// TIA Portal project "Practica3AD21" (V16)

(* hardware
DEVICE "S7300/ET200M station_1"  S7-300 station
   slot 0: "Rail_0"  Rail  6ES7 390-1***0-0AA0
   slot 2: "PLC_1"  CPU 314  6ES7 314-1AG13-0AB0  V2.6
      slot 0: "MPI interface_1"  X1
*)

// ===== PLC "PLC_1"  CPU 314 =====

VAR_GLOBAL   // PLC tag table "Memorias"
   "E0" AT %M0.0 : Bool;   // Esperando a que haya pieza en almacen
   "E1" AT %M0.1 : Bool;   // Avanzando pieza
   "E2" AT %M0.2 : Bool;   // Primera ronda deteccion
   "E3" AT %M0.3 : Bool;   // Primera ronda ninguno
   "E4" AT %M0.4 : Bool;   // Primera ronda ambos
   "E5" AT %M0.5 : Bool;   // Primera ronda alguno
   "E6" AT %M0.6 : Bool;   // Pieza Tipo 1
   "E7" AT %M0.7 : Bool;   // Pieza Tipo 2
   "E8" AT %M1.0 : Bool;   // Pieza Tipo 3
   "E9" AT %M1.1 : Bool;   // Pieza Tipo 4
   "E10" AT %M1.6 : Bool;   // Extraer Piston 1
   "E11" AT %M1.7 : Bool;   // Extraer Piston 2
   "E12" AT %M2.0 : Bool;   // Extraer Piston 3
   "E13" AT %M2.1 : Bool;   // Contraer Piston 1
   "E14" AT %M2.2 : Bool;   // Contraer Piston 2
   "E15" AT %M2.3 : Bool;   // Contraer Piston 3
   "E16" AT %M2.4 : Bool;   // Pieza 1 Termina
   "E17" AT %M2.5 : Bool;   // Pieza 2 Termina
   "E18" AT %M2.6 : Bool;   // Pieza 3 Termina
   "E19" AT %M2.7 : Bool;   // Pieza 4 Termina
   "E20" AT %M3.0 : Bool;   // Detener Programa
END_VAR

VAR_GLOBAL   // PLC tag table "Salidas"
   "Chain" AT %Q11.0 : Bool;
   "Belt" AT %Q11.1 : Bool;
   "P1toWork" AT %Q11.2 : Bool;
   "P1toHome" AT %Q11.3 : Bool;
   "P2toWork" AT %Q11.4 : Bool;
   "P2toHome" AT %Q11.5 : Bool;
   "P3toWork" AT %Q11.6 : Bool;
   "P3toHome" AT %Q11.7 : Bool;
END_VAR

VAR_GLOBAL   // PLC tag table "Entradas"
   "P3inWork" AT %I10.0 : Bool;   // NC
   "P3inHome" AT %I10.1 : Bool;   // NC
   "P3engaged" AT %I10.2 : Bool;   // NO
   "RStation1" AT %I10.3 : Bool;   // NO
   "RStation2" AT %I10.4 : Bool;   // NO
   "Lightbarrier" AT %I10.5 : Bool;   // NC
   "inPlace3" AT %I10.6 : Bool;   // NO
   "inPlace4" AT %I10.7 : Bool;   // NO
   "P1inWork" AT %I11.0 : Bool;   // NC
   "P1inHome" AT %I11.1 : Bool;   // NC
   "P2inWork" AT %I11.2 : Bool;   // NC
   "P2inHome" AT %I11.3 : Bool;   // NC
   "P1engaged" AT %I11.4 : Bool;   // NO
   "P2engaged" AT %I11.5 : Bool;   // NO
   "inPlace1" AT %I11.6 : Bool;   // NO
   "inPlace2" AT %I11.7 : Bool;   // NO
   "chainMagnet" AT %I13.6 : Bool;   // NO
   "STOP" AT %I13.7 : Bool;   // NO
   "START" AT %I13.5 : Bool;   // NO
END_VAR

// folder: SystemBlocksFolder/ReportSystemErrorFolder

DATA_BLOCK "RSE_DIAGNOSTIC_STATUS_DB"   // DB127
TITLE = Report System Error Diagnostic Block
{ S7_Optimized_Access := 'FALSE' }
AUTHOR : SIMATIC
FAMILY : RSEDIAG
NAME : RSE7
VERSION : 1.0
// This DB is part of report system error and will be updated by the RSE FB.
//  It is an interface for support of system diagnosis via the CPU web server.
   VAR
      Directory : Struct
         D_Version : Word := WORD#16#0100;   // Version that supports RSE
         D_pGlobalState : Word := WORD#16#0010;   // Byte offset to the start of the "GlobalState" section
         D_pQuery : Word := WORD#16#0014;   // Byte offset to the start of the "Query" section
         D_pComponent : Word := WORD#16#0020;   // Byte offset to the start of the "Component" section
         D_pError : Word := WORD#16#0024;   // Byte offset to the start of the "Error" section
         D_pState : Word := WORD#16#0028;   // Byte offset to the start of the "State" section
         D_pAlarm : Word := WORD#16#005A;   // Byte offset to the start of the "Alarm" section
         D_pSubComponent : Word := WORD#16#0082;   // Byte offset to the start of the "Subcomponent" section
      END_STRUCT;
      GlobalState : Struct
         G_EventCount : Word := WORD#16#0000;   // ID of the last event (counter)
         G_StartReporting : Bool := FALSE;   // Startup evaluation running
      END_STRUCT;
      Query : Struct
         Q_ClientID_User : DWord := DWORD#16#0000_0000;   // ID of the client
         Q_ClientID_Intern : DWord := DWORD#16#0000_0000;   // ID of the client (internal)
         Q_WithSubComponent : Bool := FALSE;   // With/without status of the underlying components (slower)
         Q_SubComponentAlarm : Bool := FALSE;   // AS-iMaster gibt AS-iSlave Alarme zurück
         Q_Reserved2 : Bool := FALSE;   // Reserved
         Q_Reserved3 : Bool := FALSE;   // Reserved
         Q_Reserved4 : Bool := FALSE;   // Reserved
         Q_Reserved5 : Bool := FALSE;   // Reserved
         Q_Reserved6 : Bool := FALSE;   // Reserved
         Q_Reserved7 : Bool := FALSE;   // Reserved
         Q_Start : Bool := FALSE;   // Start query
         Q_Error : Byte := BYTE#16#00;   // Internal error in query
         Q_Reserved8 : Byte := BYTE#16#00;   // Reserved
      END_STRUCT;
      Component : Struct
         C_AddressMode : Byte := BYTE#16#00;   // Addressing mode of the module
         C_Reserved1 : Byte := BYTE#16#00;   // Reserved
         C_ComponentID : Word := WORD#16#0000;   // Hardware ID of the component (internal)
      END_STRUCT;
      Error : Struct
         E_ErrorNo : Word := WORD#16#0000;   // Index of the requested/actual error
         E_LastError : Bool := FALSE;   // TRUE, if E_ErrorNo contains the indes of the last error, otherwise FALSE
      END_STRUCT;
      State : Struct
         S_Hierarchy : Byte := BYTE#16#00;   // Reserved
         S_Periphery : Byte := BYTE#16#00;   // Reserved
         S_SupFault : Bool := FALSE;   // The component is not obtainable
         S_NotAvailable : Bool := FALSE;   // The component does not exist
         S_Faulty : Bool := FALSE;   // The component is disrupted; the "Alarm" section is not empty
         S_MoreErrors : Bool := FALSE;   // There are more errors than RSE can store.
         S_Maintenance1 : Bool := FALSE;   // Maintenance required is indicated
         S_Maintenance2 : Bool := FALSE;   // Maintenance demand is indicated
         S_Deactivated : Bool := FALSE;   // The component was deactivated
         S_Reserved2 : Bool := FALSE;   // Reserved
         S_SubFault : Bool := FALSE;   // An underlying component is disrupted
         S_SubMaintenance1 : Bool := FALSE;   // Maintenance required is indicated for an underlying component
         S_SubMaintenance2 : Bool := FALSE;   // Maintenance demand is indicated for an underlying component
         S_SubDeactivated : Bool := FALSE;   // At least one lower-level component is disabled
         S_Reserved4 : Bool := FALSE;   // Reserved
         S_Reserved5 : Bool := FALSE;   // Reserved
         S_Reserved6 : Bool := FALSE;   // Reserved
         S_Reserved7 : Bool := FALSE;   // Reserved
         S_TIAMS : DWord := DWORD#16#0000_0000;   // Maintenance state of the component
         S_TIAMSChannelExist : DWord := DWORD#16#0000_0000;   // Maintenance state: Configured channels
         S_TIAMSChannelOK : DWord := DWORD#16#0000_0000;   // Maintenance State: Disrupted channels
         S_ChannelCount : Word := WORD#16#0000;   // Number of channels; Valid only when Q_WithSubComponent is set
         S_ChannelVector : Array[0..255] of Bool;   // List of channels involved; Valid only when Q_WithSubComponent is set
      END_STRUCT;
      Alarm : Struct
         A_ComponentID : Word := WORD#16#0000;   // Hardware ID of the component (internal)
         A_TextID1 : Word := WORD#16#0000;   // ID of the first error text
         A_TextLexikonID1 : Word := WORD#16#0000;   // ID of the first error text lexicon
         A_HelpTextLexikonID1 : Word := WORD#16#0000;   // ID of the first help text lexicon
         A_MapTextID : Word := WORD#16#0000;   // ID of the first error text in the export file (HMI)
         A_MapHelpTextID : Word := WORD#16#0000;   // ID of the first help text in the export file (HMI)
         A_TextID2 : Word := WORD#16#0000;   // ID of the second error text
         A_TextLexikonID2 : Word := WORD#16#0000;   // ID of the second error text lexicon
         A_HelpTextLexikonID2 : Word := WORD#16#0000;   // ID of the second help text lexicon
         A_MapTextID2 : Word := WORD#16#0000;   // ID of the second error text in the export file (HMI)
         A_MapHelpTextID2 : Word := WORD#16#0000;   // ID of the second help text in the export file (HMI)
         A_AlarmID : DWord := DWORD#16#0000_0000;   // Message number
         A_ValueCount : Word := WORD#16#000C;   // Number of other occupied bytes
         A_AssociatedValue : Array[1..6] of Word;   // Associated values of the message
      END_STRUCT;
      SubComponent : Struct
         U_SubComponentCount : Word := WORD#16#0000;   // Number of underlying components
         U_SubComponentFault : Array[1..4] of Byte;   // List of status of subordinate components, 1 byte per component
      END_STRUCT;
   END_VAR
BEGIN
END_DATA_BLOCK

// folder: (top level)

FUNCTION "Secuencial" : Void   // FC1, LAD
{ S7_Optimized_Access := 'FALSE' }
VERSION : 0.1
   VAR_TEMP
      T1A : Time;
   END_VAR
   VAR_TEMP   // added for the SCL form of the ladder/FBD networks
      _w1 : Bool;
   END_VAR
BEGIN

REGION Network 1: Avanzando pieza
   // Si se detecta una pieza en el almacen y no se ha apretado STOP, mover la cadena
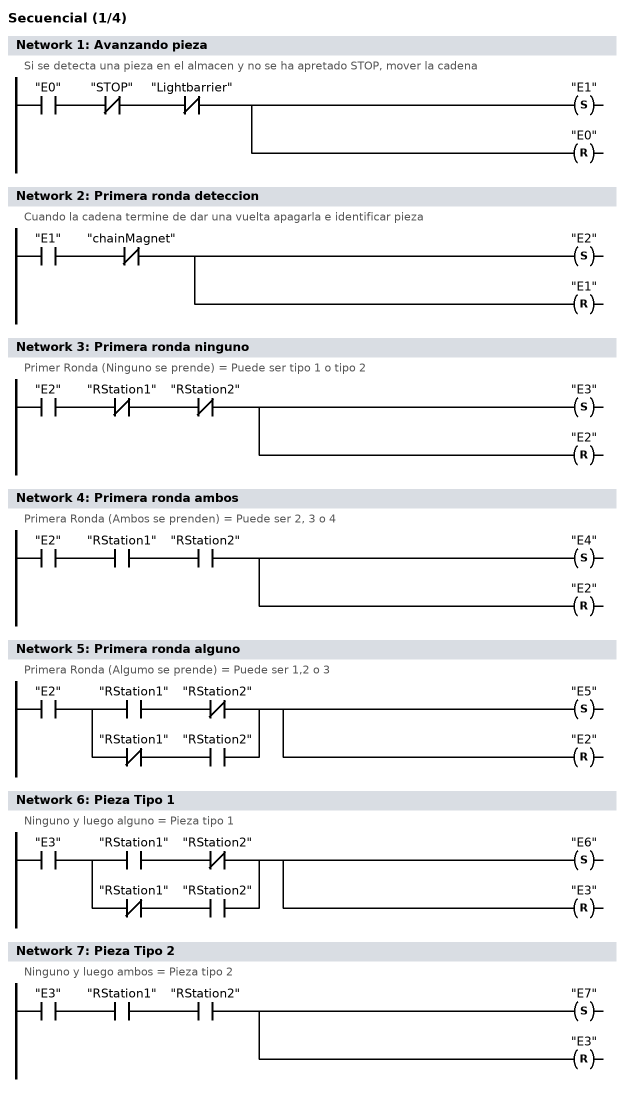
   RUNG wire#powerrail
      Contact( "E0" )
      I_Contact( "STOP" )
      I_Contact( "Lightbarrier" )
      wire#w1
      S_Coil( "E1" )
   END_RUNG
   RUNG wire#w1
      R_Coil( "E0" )
   END_RUNG
   // the same network as SCL:
   IF "E0" AND NOT "STOP" AND NOT "Lightbarrier" THEN
       "E1" := TRUE;
       "E0" := FALSE;
   END_IF;
END_REGION

REGION Network 2: Primera ronda deteccion
   // Cuando la cadena termine de dar una vuelta apagarla e identificar pieza
   RUNG wire#powerrail
      Contact( "E1" )
      I_Contact( "chainMagnet" )
      wire#w1
      S_Coil( "E2" )
   END_RUNG
   RUNG wire#w1
      R_Coil( "E1" )
   END_RUNG
   // the same network as SCL:
   IF "E1" AND NOT "chainMagnet" THEN
       "E2" := TRUE;
       "E1" := FALSE;
   END_IF;
END_REGION

REGION Network 3: Primera ronda ninguno
   // Primer Ronda (Ninguno se prende) = Puede ser tipo 1 o tipo 2
   RUNG wire#powerrail
      Contact( "E2" )
      I_Contact( "RStation1" )
      I_Contact( "RStation2" )
      wire#w1
      S_Coil( "E3" )
   END_RUNG
   RUNG wire#w1
      R_Coil( "E2" )
   END_RUNG
   // the same network as SCL:
   IF "E2" AND NOT "RStation1" AND NOT "RStation2" THEN
       "E3" := TRUE;
       "E2" := FALSE;
   END_IF;
END_REGION

REGION Network 4: Primera ronda ambos
   // Primera Ronda (Ambos se prenden) = Puede ser 2, 3 o 4
   RUNG wire#powerrail
      Contact( "E2" )
      Contact( "RStation1" )
      Contact( "RStation2" )
      wire#w1
      S_Coil( "E4" )
   END_RUNG
   RUNG wire#w1
      R_Coil( "E2" )
   END_RUNG
   // the same network as SCL:
   IF "E2" AND "RStation1" AND "RStation2" THEN
       "E4" := TRUE;
       "E2" := FALSE;
   END_IF;
END_REGION

REGION Network 5: Primera ronda alguno
   // Primera Ronda (Algumo se prende) = Puede ser 1,2 o 3
   RUNG wire#powerrail
      Contact( "E2" )
      wire#w1
      Contact( "RStation1" )
      I_Contact( "RStation2" )
      wire#w2
      S_Coil( "E5" )
   END_RUNG
   RUNG wire#w1
      I_Contact( "RStation1" )
      Contact( "RStation2" )
   END_RUNG wire#w2
   RUNG wire#w2
      R_Coil( "E2" )
   END_RUNG
   // the same network as SCL:
   IF "E2" AND (("RStation1" AND NOT "RStation2") OR (NOT "RStation1" AND "RStation2")) THEN
       "E5" := TRUE;
       "E2" := FALSE;
   END_IF;
END_REGION

REGION Network 6: Pieza Tipo 1
   // Ninguno y luego alguno = Pieza tipo 1
   RUNG wire#powerrail
      Contact( "E3" )
      wire#w1
      Contact( "RStation1" )
      I_Contact( "RStation2" )
      wire#w2
      S_Coil( "E6" )
   END_RUNG
   RUNG wire#w1
      I_Contact( "RStation1" )
      Contact( "RStation2" )
   END_RUNG wire#w2
   RUNG wire#w2
      R_Coil( "E3" )
   END_RUNG
   // the same network as SCL:
   IF "E3" AND (("RStation1" AND NOT "RStation2") OR (NOT "RStation1" AND "RStation2")) THEN
       "E6" := TRUE;
       "E3" := FALSE;
   END_IF;
END_REGION

REGION Network 7: Pieza Tipo 2
   // Ninguno y luego ambos = Pieza tipo 2
   RUNG wire#powerrail
      Contact( "E3" )
      Contact( "RStation1" )
      Contact( "RStation2" )
      wire#w1
      S_Coil( "E7" )
   END_RUNG
   RUNG wire#w1
      R_Coil( "E3" )
   END_RUNG
   // the same network as SCL:
   IF "E3" AND "RStation1" AND "RStation2" THEN
       "E7" := TRUE;
       "E3" := FALSE;
   END_IF;
END_REGION

REGION Network 8: Pieza Tipo 2
   // Ambos y luego ninguno = Pieza tipo 2
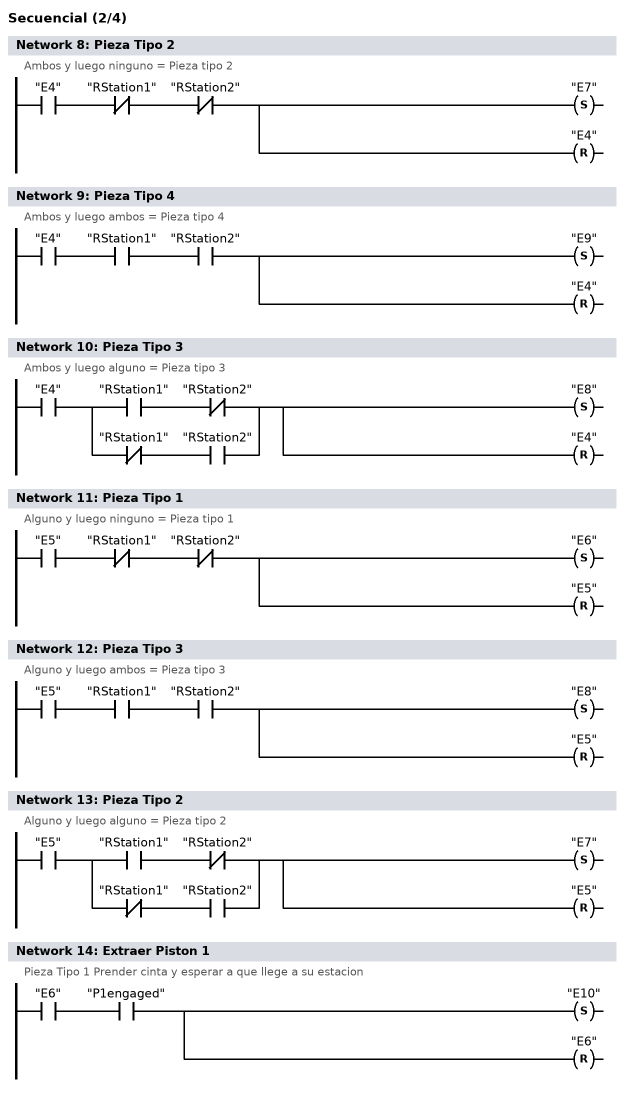
   RUNG wire#powerrail
      Contact( "E4" )
      I_Contact( "RStation1" )
      I_Contact( "RStation2" )
      wire#w1
      S_Coil( "E7" )
   END_RUNG
   RUNG wire#w1
      R_Coil( "E4" )
   END_RUNG
   // the same network as SCL:
   IF "E4" AND NOT "RStation1" AND NOT "RStation2" THEN
       "E7" := TRUE;
       "E4" := FALSE;
   END_IF;
END_REGION

REGION Network 9: Pieza Tipo 4
   // Ambos y luego ambos = Pieza tipo 4
   RUNG wire#powerrail
      Contact( "E4" )
      Contact( "RStation1" )
      Contact( "RStation2" )
      wire#w1
      S_Coil( "E9" )
   END_RUNG
   RUNG wire#w1
      R_Coil( "E4" )
   END_RUNG
   // the same network as SCL:
   IF "E4" AND "RStation1" AND "RStation2" THEN
       "E9" := TRUE;
       "E4" := FALSE;
   END_IF;
END_REGION

REGION Network 10: Pieza Tipo 3
   // Ambos y luego alguno = Pieza tipo 3
   RUNG wire#powerrail
      Contact( "E4" )
      wire#w1
      Contact( "RStation1" )
      I_Contact( "RStation2" )
      wire#w2
      S_Coil( "E8" )
   END_RUNG
   RUNG wire#w1
      I_Contact( "RStation1" )
      Contact( "RStation2" )
   END_RUNG wire#w2
   RUNG wire#w2
      R_Coil( "E4" )
   END_RUNG
   // the same network as SCL:
   IF "E4" AND (("RStation1" AND NOT "RStation2") OR (NOT "RStation1" AND "RStation2")) THEN
       "E8" := TRUE;
       "E4" := FALSE;
   END_IF;
END_REGION

REGION Network 11: Pieza Tipo 1
   // Alguno y luego ninguno = Pieza tipo 1
   RUNG wire#powerrail
      Contact( "E5" )
      I_Contact( "RStation1" )
      I_Contact( "RStation2" )
      wire#w1
      S_Coil( "E6" )
   END_RUNG
   RUNG wire#w1
      R_Coil( "E5" )
   END_RUNG
   // the same network as SCL:
   IF "E5" AND NOT "RStation1" AND NOT "RStation2" THEN
       "E6" := TRUE;
       "E5" := FALSE;
   END_IF;
END_REGION

REGION Network 12: Pieza Tipo 3
   // Alguno y luego ambos = Pieza tipo 3
   RUNG wire#powerrail
      Contact( "E5" )
      Contact( "RStation1" )
      Contact( "RStation2" )
      wire#w1
      S_Coil( "E8" )
   END_RUNG
   RUNG wire#w1
      R_Coil( "E5" )
   END_RUNG
   // the same network as SCL:
   IF "E5" AND "RStation1" AND "RStation2" THEN
       "E8" := TRUE;
       "E5" := FALSE;
   END_IF;
END_REGION

REGION Network 13: Pieza Tipo 2
   // Alguno y luego alguno = Pieza tipo 2
   RUNG wire#powerrail
      Contact( "E5" )
      wire#w1
      Contact( "RStation1" )
      I_Contact( "RStation2" )
      wire#w2
      S_Coil( "E7" )
   END_RUNG
   RUNG wire#w1
      I_Contact( "RStation1" )
      Contact( "RStation2" )
   END_RUNG wire#w2
   RUNG wire#w2
      R_Coil( "E5" )
   END_RUNG
   // the same network as SCL:
   IF "E5" AND (("RStation1" AND NOT "RStation2") OR (NOT "RStation1" AND "RStation2")) THEN
       "E7" := TRUE;
       "E5" := FALSE;
   END_IF;
END_REGION

REGION Network 14: Extraer Piston 1
   // Pieza Tipo 1 Prender cinta y esperar a que llege a su estacion
   RUNG wire#powerrail
      Contact( "E6" )
      Contact( "P1engaged" )
      wire#w1
      S_Coil( "E10" )
   END_RUNG
   RUNG wire#w1
      R_Coil( "E6" )
   END_RUNG
   // the same network as SCL:
   IF "E6" AND "P1engaged" THEN
       "E10" := TRUE;
       "E6" := FALSE;
   END_IF;
END_REGION

REGION Network 15: Extraer Piston 2
   // Pieza Tipo 2 Prender cinta y esperar a que llege a su estacion
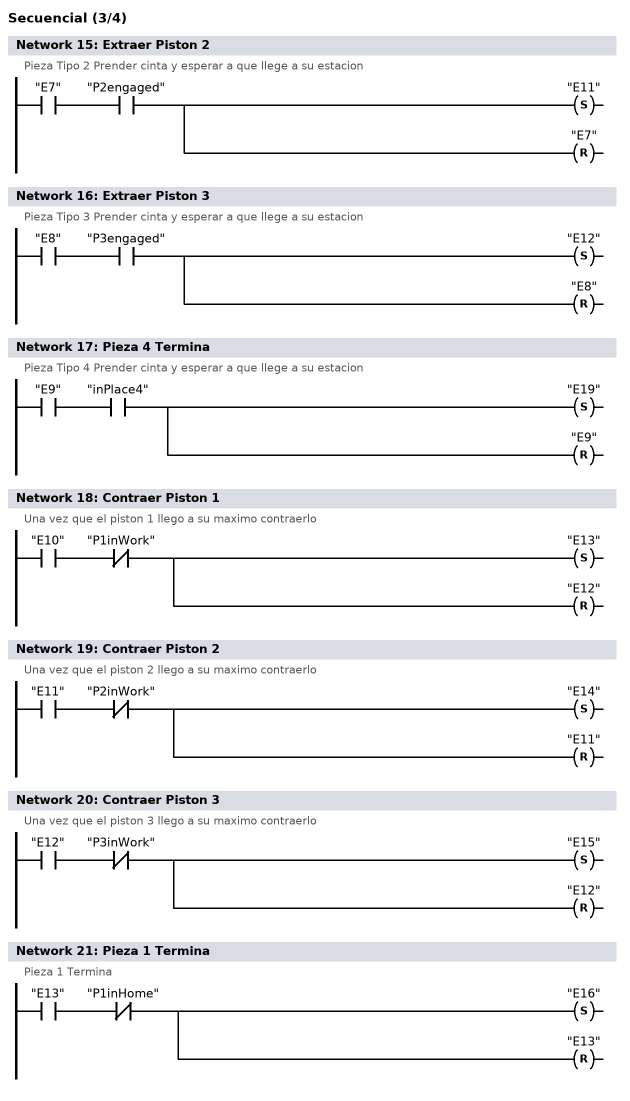
   RUNG wire#powerrail
      Contact( "E7" )
      Contact( "P2engaged" )
      wire#w1
      S_Coil( "E11" )
   END_RUNG
   RUNG wire#w1
      R_Coil( "E7" )
   END_RUNG
   // the same network as SCL:
   IF "E7" AND "P2engaged" THEN
       "E11" := TRUE;
       "E7" := FALSE;
   END_IF;
END_REGION

REGION Network 16: Extraer Piston 3
   // Pieza Tipo 3 Prender cinta y esperar a que llege a su estacion
   RUNG wire#powerrail
      Contact( "E8" )
      Contact( "P3engaged" )
      wire#w1
      S_Coil( "E12" )
   END_RUNG
   RUNG wire#w1
      R_Coil( "E8" )
   END_RUNG
   // the same network as SCL:
   IF "E8" AND "P3engaged" THEN
       "E12" := TRUE;
       "E8" := FALSE;
   END_IF;
END_REGION

REGION Network 17: Pieza 4 Termina
   // Pieza Tipo 4 Prender cinta y esperar a que llege a su estacion
   RUNG wire#powerrail
      Contact( "E9" )
      Contact( "inPlace4" )
      wire#w1
      S_Coil( "E19" )
   END_RUNG
   RUNG wire#w1
      R_Coil( "E9" )
   END_RUNG
   // the same network as SCL:
   IF "E9" AND "inPlace4" THEN
       "E19" := TRUE;
       "E9" := FALSE;
   END_IF;
END_REGION

REGION Network 18: Contraer Piston 1
   // Una vez que el piston 1 llego a su maximo contraerlo
   RUNG wire#powerrail
      Contact( "E10" )
      I_Contact( "P1inWork" )
      wire#w1
      S_Coil( "E13" )
   END_RUNG
   RUNG wire#w1
      R_Coil( "E12" )
   END_RUNG
   // the same network as SCL:
   IF "E10" AND NOT "P1inWork" THEN
       "E13" := TRUE;
       "E12" := FALSE;
   END_IF;
END_REGION

REGION Network 19: Contraer Piston 2
   // Una vez que el piston 2 llego a su maximo contraerlo
   RUNG wire#powerrail
      Contact( "E11" )
      I_Contact( "P2inWork" )
      wire#w1
      S_Coil( "E14" )
   END_RUNG
   RUNG wire#w1
      R_Coil( "E11" )
   END_RUNG
   // the same network as SCL:
   IF "E11" AND NOT "P2inWork" THEN
       "E14" := TRUE;
       "E11" := FALSE;
   END_IF;
END_REGION

REGION Network 20: Contraer Piston 3
   // Una vez que el piston 3 llego a su maximo contraerlo
   RUNG wire#powerrail
      Contact( "E12" )
      I_Contact( "P3inWork" )
      wire#w1
      S_Coil( "E15" )
   END_RUNG
   RUNG wire#w1
      R_Coil( "E12" )
   END_RUNG
   // the same network as SCL:
   IF "E12" AND NOT "P3inWork" THEN
       "E15" := TRUE;
       "E12" := FALSE;
   END_IF;
END_REGION

REGION Network 21: Pieza 1 Termina
   // Pieza 1 Termina
   RUNG wire#powerrail
      Contact( "E13" )
      I_Contact( "P1inHome" )
      wire#w1
      S_Coil( "E16" )
   END_RUNG
   RUNG wire#w1
      R_Coil( "E13" )
   END_RUNG
   // the same network as SCL:
   IF "E13" AND NOT "P1inHome" THEN
       "E16" := TRUE;
       "E13" := FALSE;
   END_IF;
END_REGION

REGION Network 22: Pieza 2 Termina
   // Pieza 2 Termina
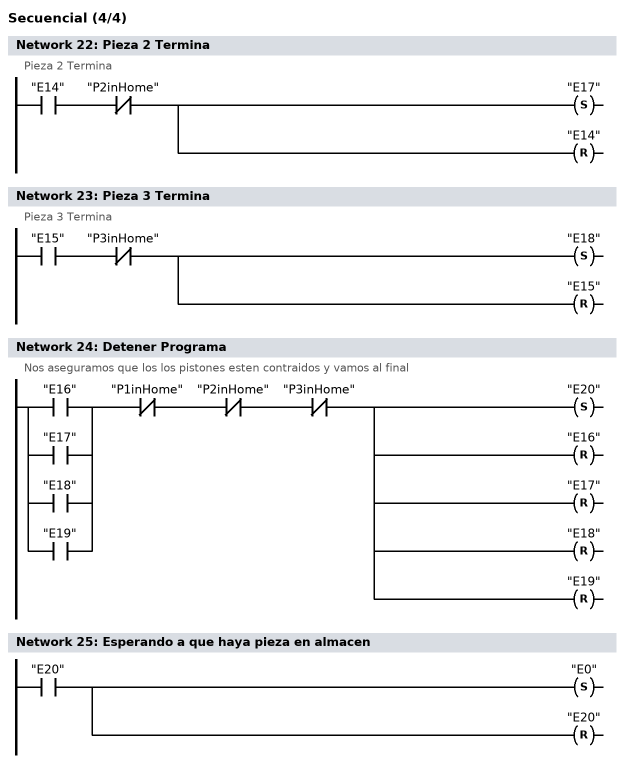
   RUNG wire#powerrail
      Contact( "E14" )
      I_Contact( "P2inHome" )
      wire#w1
      S_Coil( "E17" )
   END_RUNG
   RUNG wire#w1
      R_Coil( "E14" )
   END_RUNG
   // the same network as SCL:
   IF "E14" AND NOT "P2inHome" THEN
       "E17" := TRUE;
       "E14" := FALSE;
   END_IF;
END_REGION

REGION Network 23: Pieza 3 Termina
   // Pieza 3 Termina
   RUNG wire#powerrail
      Contact( "E15" )
      I_Contact( "P3inHome" )
      wire#w1
      S_Coil( "E18" )
   END_RUNG
   RUNG wire#w1
      R_Coil( "E15" )
   END_RUNG
   // the same network as SCL:
   IF "E15" AND NOT "P3inHome" THEN
       "E18" := TRUE;
       "E15" := FALSE;
   END_IF;
END_REGION

REGION Network 24: Detener Programa
   // Nos aseguramos que los los pistones esten contraidos y vamos al final
   RUNG wire#powerrail
      Contact( "E16" )
      wire#w1
      I_Contact( "P1inHome" )
      I_Contact( "P2inHome" )
      I_Contact( "P3inHome" )
      wire#w2
      S_Coil( "E20" )
   END_RUNG
   RUNG wire#powerrail
      Contact( "E17" )
   END_RUNG wire#w1
   RUNG wire#powerrail
      Contact( "E18" )
   END_RUNG wire#w1
   RUNG wire#powerrail
      Contact( "E19" )
   END_RUNG wire#w1
   RUNG wire#w2
      R_Coil( "E16" )
   END_RUNG
   RUNG wire#w2
      R_Coil( "E17" )
   END_RUNG
   RUNG wire#w2
      R_Coil( "E18" )
   END_RUNG
   RUNG wire#w2
      R_Coil( "E19" )
   END_RUNG
   // the same network as SCL:
   IF ("E16" OR "E17" OR "E18" OR "E19") AND NOT "P1inHome" AND NOT "P2inHome" AND NOT "P3inHome" THEN
       "E20" := TRUE;
   END_IF;
   #_w1 := ("E16" OR "E17" OR "E18" OR "E19") AND NOT "P1inHome" AND NOT "P2inHome" AND NOT "P3inHome";
   IF #_w1 THEN
       "E16" := FALSE;
       "E17" := FALSE;
       "E18" := FALSE;
       "E19" := FALSE;
   END_IF;
END_REGION

REGION Network 25: Esperando a que haya pieza en almacen
   RUNG wire#powerrail
      Contact( "E20" )
      wire#w1
      S_Coil( "E0" )
   END_RUNG
   RUNG wire#w1
      R_Coil( "E20" )
   END_RUNG
   // the same network as SCL:
   IF "E20" THEN
       "E0" := TRUE;
       "E20" := FALSE;
   END_IF;
END_REGION
END_FUNCTION

FUNCTION "Combinacional" : Void   // FC2, LAD
{ S7_Optimized_Access := 'FALSE' }
VERSION : 0.1
BEGIN

REGION Network 1
   // Cuando inicia el programa todo esta apagado
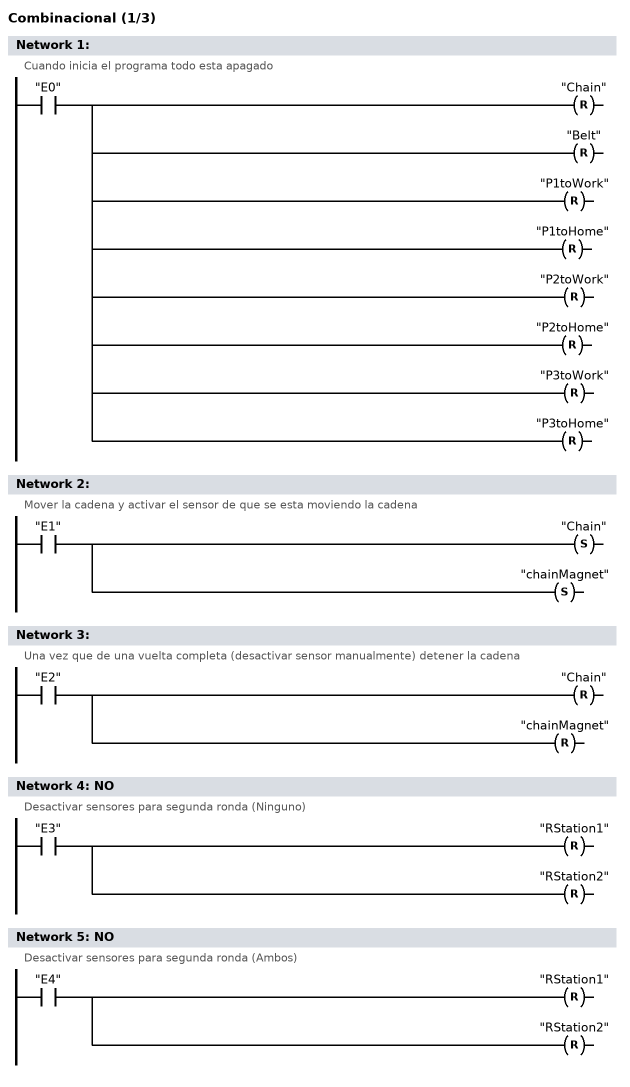
   RUNG wire#powerrail
      Contact( "E0" )
      wire#w1
      R_Coil( "Chain" )
   END_RUNG
   RUNG wire#w1
      R_Coil( "Belt" )
   END_RUNG
   RUNG wire#w1
      R_Coil( "P1toWork" )
   END_RUNG
   RUNG wire#w1
      R_Coil( "P1toHome" )
   END_RUNG
   RUNG wire#w1
      R_Coil( "P2toWork" )
   END_RUNG
   RUNG wire#w1
      R_Coil( "P2toHome" )
   END_RUNG
   RUNG wire#w1
      R_Coil( "P3toWork" )
   END_RUNG
   RUNG wire#w1
      R_Coil( "P3toHome" )
   END_RUNG
   // the same network as SCL:
   IF "E0" THEN
       "Chain" := FALSE;
       "Belt" := FALSE;
       "P1toWork" := FALSE;
       "P1toHome" := FALSE;
       "P2toWork" := FALSE;
       "P2toHome" := FALSE;
       "P3toWork" := FALSE;
       "P3toHome" := FALSE;
   END_IF;
END_REGION

REGION Network 2
   // Mover la cadena y activar el sensor de que se esta moviendo la cadena
   RUNG wire#powerrail
      Contact( "E1" )
      wire#w1
      S_Coil( "Chain" )
   END_RUNG
   RUNG wire#w1
      S_Coil( "chainMagnet" )
   END_RUNG
   // the same network as SCL:
   IF "E1" THEN
       "Chain" := TRUE;
       "chainMagnet" := TRUE;
   END_IF;
END_REGION

REGION Network 3
   // Una vez que de una vuelta completa (desactivar sensor manualmente) detener la cadena
   RUNG wire#powerrail
      Contact( "E2" )
      wire#w1
      R_Coil( "Chain" )
   END_RUNG
   RUNG wire#w1
      R_Coil( "chainMagnet" )
   END_RUNG
   // the same network as SCL:
   IF "E2" THEN
       "Chain" := FALSE;
       "chainMagnet" := FALSE;
   END_IF;
END_REGION

REGION Network 4: NO
   // Desactivar sensores para segunda ronda (Ninguno)
   RUNG wire#powerrail
      Contact( "E3" )
      wire#w1
      R_Coil( "RStation1" )
   END_RUNG
   RUNG wire#w1
      R_Coil( "RStation2" )
   END_RUNG
   // the same network as SCL:
   IF "E3" THEN
       "RStation1" := FALSE;
       "RStation2" := FALSE;
   END_IF;
END_REGION

REGION Network 5: NO
   // Desactivar sensores para segunda ronda (Ambos)
   RUNG wire#powerrail
      Contact( "E4" )
      wire#w1
      R_Coil( "RStation1" )
   END_RUNG
   RUNG wire#w1
      R_Coil( "RStation2" )
   END_RUNG
   // the same network as SCL:
   IF "E4" THEN
       "RStation1" := FALSE;
       "RStation2" := FALSE;
   END_IF;
END_REGION

REGION Network 6: NO
   // Desactivar sensores para segunda ronda (Alguno)
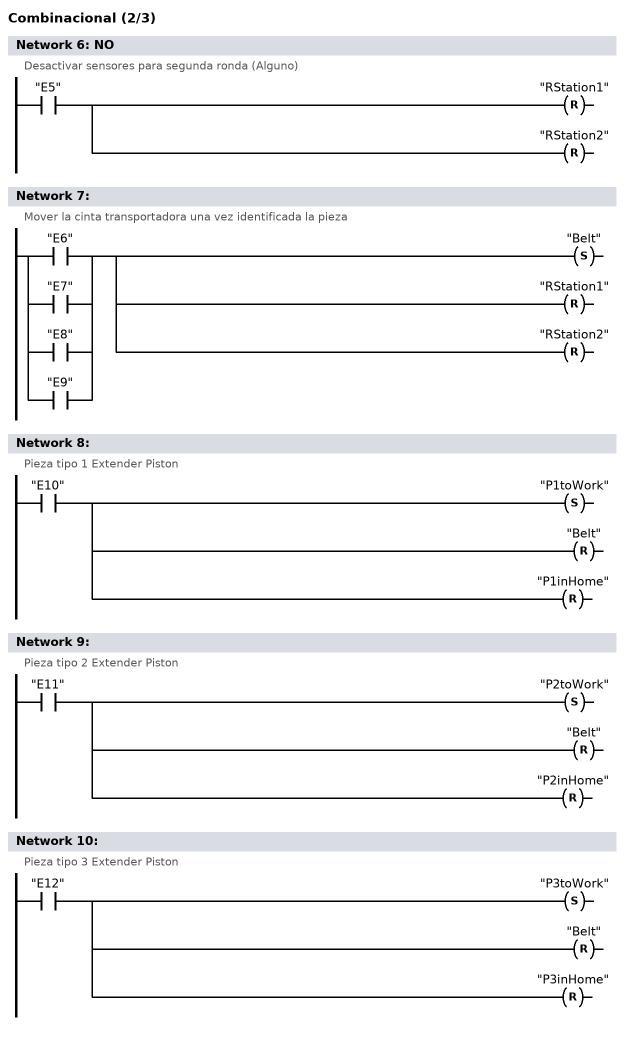
   RUNG wire#powerrail
      Contact( "E5" )
      wire#w1
      R_Coil( "RStation1" )
   END_RUNG
   RUNG wire#w1
      R_Coil( "RStation2" )
   END_RUNG
   // the same network as SCL:
   IF "E5" THEN
       "RStation1" := FALSE;
       "RStation2" := FALSE;
   END_IF;
END_REGION

REGION Network 7
   // Mover la cinta transportadora una vez identificada la pieza
   RUNG wire#powerrail
      Contact( "E6" )
      wire#w1
      S_Coil( "Belt" )
   END_RUNG
   RUNG wire#powerrail
      Contact( "E7" )
   END_RUNG wire#w1
   RUNG wire#powerrail
      Contact( "E8" )
   END_RUNG wire#w1
   RUNG wire#powerrail
      Contact( "E9" )
   END_RUNG wire#w1
   RUNG wire#w1
      R_Coil( "RStation1" )
   END_RUNG
   RUNG wire#w1
      R_Coil( "RStation2" )
   END_RUNG
   // the same network as SCL:
   IF "E6" OR "E7" OR "E8" OR "E9" THEN
       "Belt" := TRUE;
       "RStation1" := FALSE;
       "RStation2" := FALSE;
   END_IF;
END_REGION

REGION Network 8
   // Pieza tipo 1 Extender Piston
   RUNG wire#powerrail
      Contact( "E10" )
      wire#w1
      S_Coil( "P1toWork" )
   END_RUNG
   RUNG wire#w1
      R_Coil( "Belt" )
   END_RUNG
   RUNG wire#w1
      R_Coil( "P1inHome" )
   END_RUNG
   // the same network as SCL:
   IF "E10" THEN
       "P1toWork" := TRUE;
       "Belt" := FALSE;
       "P1inHome" := FALSE;
   END_IF;
END_REGION

REGION Network 9
   // Pieza tipo 2 Extender Piston
   RUNG wire#powerrail
      Contact( "E11" )
      wire#w1
      S_Coil( "P2toWork" )
   END_RUNG
   RUNG wire#w1
      R_Coil( "Belt" )
   END_RUNG
   RUNG wire#w1
      R_Coil( "P2inHome" )
   END_RUNG
   // the same network as SCL:
   IF "E11" THEN
       "P2toWork" := TRUE;
       "Belt" := FALSE;
       "P2inHome" := FALSE;
   END_IF;
END_REGION

REGION Network 10
   // Pieza tipo 3 Extender Piston
   RUNG wire#powerrail
      Contact( "E12" )
      wire#w1
      S_Coil( "P3toWork" )
   END_RUNG
   RUNG wire#w1
      R_Coil( "Belt" )
   END_RUNG
   RUNG wire#w1
      R_Coil( "P3inHome" )
   END_RUNG
   // the same network as SCL:
   IF "E12" THEN
       "P3toWork" := TRUE;
       "Belt" := FALSE;
       "P3inHome" := FALSE;
   END_IF;
END_REGION

REGION Network 11
   // Pieza tipo 1 Contraer Piston
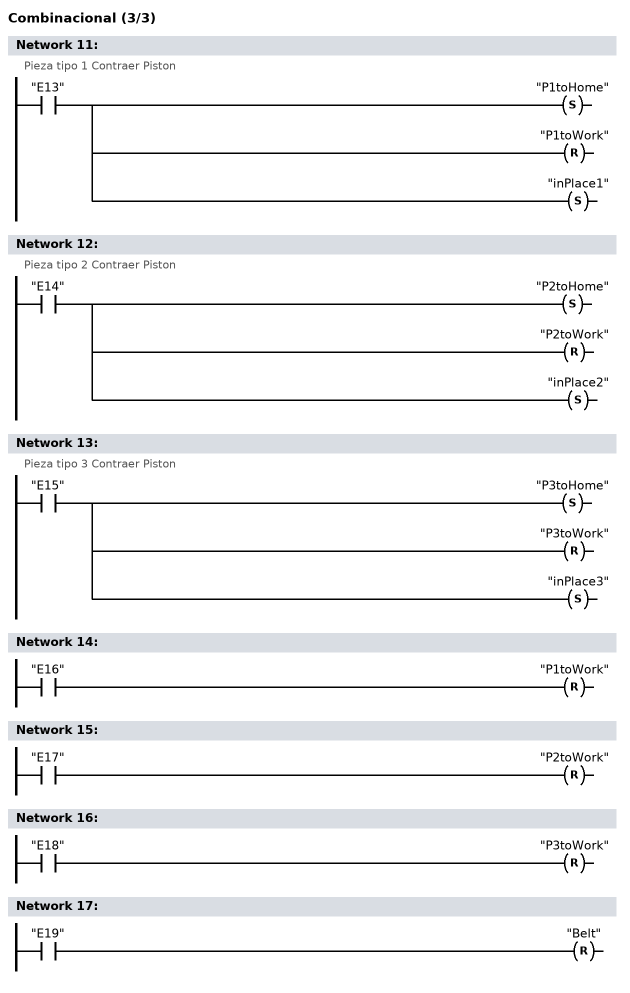
   RUNG wire#powerrail
      Contact( "E13" )
      wire#w1
      S_Coil( "P1toHome" )
   END_RUNG
   RUNG wire#w1
      R_Coil( "P1toWork" )
   END_RUNG
   RUNG wire#w1
      S_Coil( "inPlace1" )
   END_RUNG
   // the same network as SCL:
   IF "E13" THEN
       "P1toHome" := TRUE;
       "P1toWork" := FALSE;
       "inPlace1" := TRUE;
   END_IF;
END_REGION

REGION Network 12
   // Pieza tipo 2 Contraer Piston
   RUNG wire#powerrail
      Contact( "E14" )
      wire#w1
      S_Coil( "P2toHome" )
   END_RUNG
   RUNG wire#w1
      R_Coil( "P2toWork" )
   END_RUNG
   RUNG wire#w1
      S_Coil( "inPlace2" )
   END_RUNG
   // the same network as SCL:
   IF "E14" THEN
       "P2toHome" := TRUE;
       "P2toWork" := FALSE;
       "inPlace2" := TRUE;
   END_IF;
END_REGION

REGION Network 13
   // Pieza tipo 3 Contraer Piston
   RUNG wire#powerrail
      Contact( "E15" )
      wire#w1
      S_Coil( "P3toHome" )
   END_RUNG
   RUNG wire#w1
      R_Coil( "P3toWork" )
   END_RUNG
   RUNG wire#w1
      S_Coil( "inPlace3" )
   END_RUNG
   // the same network as SCL:
   IF "E15" THEN
       "P3toHome" := TRUE;
       "P3toWork" := FALSE;
       "inPlace3" := TRUE;
   END_IF;
END_REGION

REGION Network 14
   RUNG wire#powerrail
      Contact( "E16" )
      R_Coil( "P1toWork" )
   END_RUNG
   // the same network as SCL:
   IF "E16" THEN "P1toWork" := FALSE; END_IF;
END_REGION

REGION Network 15
   RUNG wire#powerrail
      Contact( "E17" )
      R_Coil( "P2toWork" )
   END_RUNG
   // the same network as SCL:
   IF "E17" THEN "P2toWork" := FALSE; END_IF;
END_REGION

REGION Network 16
   RUNG wire#powerrail
      Contact( "E18" )
      R_Coil( "P3toWork" )
   END_RUNG
   // the same network as SCL:
   IF "E18" THEN "P3toWork" := FALSE; END_IF;
END_REGION

REGION Network 17
   RUNG wire#powerrail
      Contact( "E19" )
      R_Coil( "Belt" )
   END_RUNG
   // the same network as SCL:
   IF "E19" THEN "Belt" := FALSE; END_IF;
END_REGION
END_FUNCTION

ORGANIZATION_BLOCK "Main"   // OB1, LAD
TITLE = "Main Program Sweep (Cycle)"
{ S7_Optimized_Access := 'FALSE' }
VERSION : 0.1
   VAR_TEMP
      OB1_EV_CLASS : Byte;   // Bits 0-3 = 1 (Coming event), Bits 4-7 = 1 (Event class 1)
      OB1_SCAN_1 : Byte;   // 1 (Cold restart scan 1 of OB 1), 3 (Scan 2-n of OB 1)
      OB1_PRIORITY : Byte;   // Priority of OB Execution
      OB1_OB_NUMBR : Byte;   // 1 (Organization block 1, OB1)
      OB1_RESERVED_1 : Byte;   // Reserved for system
      OB1_RESERVED_2 : Byte;   // Reserved for system
      OB1_PREV_CYCLE : Int;   // Cycle time of previous OB1 scan (milliseconds)
      OB1_MIN_CYCLE : Int;   // Minimum cycle time of OB1 (milliseconds)
      OB1_MAX_CYCLE : Int;   // Maximum cycle time of OB1 (milliseconds)
      OB1_DATE_TIME : Date_And_Time;   // Date and time OB1 started
   END_VAR
BEGIN

REGION Network 1: Esperando a que haya pieza en almacen
   // Si se aprieta el boton de inicio comienza el programa
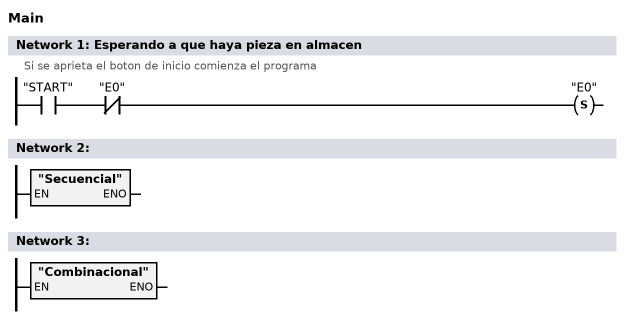
   RUNG wire#powerrail
      Contact( "START" )
      I_Contact( "E0" )
      S_Coil( "E0" )
   END_RUNG
   // the same network as SCL:
   IF "START" AND NOT "E0" THEN "E0" := TRUE; END_IF;
END_REGION

REGION Network 2
   RUNG wire#powerrail
      "Secuencial"()
   END_RUNG
   // the same network as SCL:
   "Secuencial"();
END_REGION

REGION Network 3
   RUNG wire#powerrail
      "Combinacional"()
   END_RUNG
   // the same network as SCL:
   "Combinacional"();
END_REGION

REGION Network 5 (STL): Call system diagnostics block
         CALL  "RSE_FB", "RSE_DB";
END_REGION
END_ORGANIZATION_BLOCK

ORGANIZATION_BLOCK "I/O_FLT1"   // OB82, STL
TITLE = "I/O Point Fault"
{ S7_Optimized_Access := 'FALSE' }
VERSION : 0.1
   VAR_TEMP
      OB82_EV_CLASS : Byte;   // 16#39, Event class 3, Entering event state, Internal fault event
      OB82_FLT_ID : Byte;   // 16#XX, Fault identifcation code
      OB82_PRIORITY : Byte;   // Priority of OB Execution
      OB82_OB_NUMBR : Byte;   // 82 (Organization block 82, OB82)
      OB82_RESERVED_1 : Byte;   // Reserved for system
      OB82_IO_FLAG : Byte;   // Input (01010100), Output (01010101)
      OB82_MDL_ADDR : Word;   // Base address of module with fault
      OB82_MDL_DEFECT : Bool;   // Module defective
      OB82_INT_FAULT : Bool;   // Internal fault
      OB82_EXT_FAULT : Bool;   // External fault
      OB82_PNT_INFO : Bool;   // Point information
      OB82_EXT_VOLTAGE : Bool;   // External voltage low
      OB82_FLD_CONNCTR : Bool;   // Field wiring connector missing
      OB82_NO_CONFIG : Bool;   // Module has no configuration data
      OB82_CONFIG_ERR : Bool;   // Module has configuration error
      OB82_MDL_TYPE : Byte;   // Type of module
      OB82_SUB_MDL_ERR : Bool;   // Sub-Module is missing or has error
      OB82_COMM_FAULT : Bool;   // Communication fault
      OB82_MDL_STOP : Bool;   // Module is stopped
      OB82_WTCH_DOG_FLT : Bool;   // Watch dog timer stopped module
      OB82_INT_PS_FLT : Bool;   // Internal power supply fault
      OB82_PRIM_BATT_FLT : Bool;   // Primary battery is in fault
      OB82_BCKUP_BATT_FLT : Bool;   // Backup battery is in fault
      OB82_RESERVED_2 : Bool;   // Reserved for system
      OB82_RACK_FLT : Bool;   // Rack fault, only for bus interface module
      OB82_PROC_FLT : Bool;   // Processor fault
      OB82_EPROM_FLT : Bool;   // EPROM fault
      OB82_RAM_FLT : Bool;   // RAM fault
      OB82_ADU_FLT : Bool;   // ADU fault
      OB82_FUSE_FLT : Bool;   // Fuse fault
      OB82_HW_INTR_FLT : Bool;   // Hardware interupt input in fault
      OB82_RESERVED_3 : Bool;   // Reserved for system
      OB82_DATE_TIME : Date_And_Time;   // Date and time OB82 started
   END_VAR
BEGIN

REGION Network 1: Call system diagnostics block
         CALL  "RSE_FB", "RSE_DB";
END_REGION
END_ORGANIZATION_BLOCK

ORGANIZATION_BLOCK "OBNL_FLT"   // OB85, STL
TITLE = "Organization Block (OB) Not Loaded Fault"
{ S7_Optimized_Access := 'FALSE' }
   VAR_TEMP
      OB85_EV_CLASS : Byte;   // 16#35 Event class 3
      OB85_FLT_ID : Byte;   // 16#XX, Fault identification code
      OB85_PRIORITY : Byte;   // Priority of OB Execution
      OB85_OB_NUMBR : Byte;   // 85 (Organization block 85, OB85)
      OB85_RESERVED_1 : Byte;   // Reserved for system
      OB85_RESERVED_2 : Byte;   // Reserved for system
      OB85_RESERVED_3 : Int;   // Reserved for system
      OB85_ERR_EV_CLASS : Byte;   // Class of event causing error
      OB85_ERR_EV_NUM : Byte;   // Number of event causing error
      OB85_OB_PRIOR : Byte;   // Priority of OB causing error
      OB85_OB_NUM : Byte;   // Number of OB causing error
      OB85_DATE_TIME : Date_And_Time;   // Date and time OB85 started
   END_VAR
BEGIN

REGION Network 1
         L     b#16#A1;  //
         L     #OB85_FLT_ID;
         ==I;
         JC    K_OB;
         L     b#16#A2;  //
         ==I;
         JC    K_OB;
         L     b#16#A3;  //
         L     #OB85_FLT_ID;
         ==I;
         JC    K_B;
         JU    F_PA;
END_REGION

REGION Network 2
   K_OB: JU    STOP;
         JU    ENDE;
END_REGION

REGION Network 3
   K_B:  JU    STOP;
         JU    ENDE;
END_REGION

REGION Network 4
   F_PA: NOP   0;
         JU    ENDE;
END_REGION

REGION Network 5
   STOP: CALL  STP;
END_REGION

REGION Network 6

   //

   ENDE: NOP   0;
END_REGION
END_ORGANIZATION_BLOCK